(* Schneider Machine Expert - Basic project ControlPlantaCuchildeo, file version 2.6.0.0 *)
(* CompanyInformations: Name=DMA ENERGIA *)
(* ProjectInformations: Name=CONTROL POSICION SERVO, Description=Cuchildeo *)

HARDWARE
  Cpu 0: TM221CE40T
  ModuleExtensionObject 0: TM3AM6/G
  EthernetConfiguration: NetworkName=M221, IpAllocationMode=FixedAddress, IpAddress=192.168.10.132, SubnetMask=255.255.255.0
  SerialLineConfiguration: Baud=Baud19200, Parity=ParityEven, DataBits=DataBits8, StopBits=StopBits1, PhysicalMedium=PhysicalMediumRs485, SlaveId=1, Addressing=SlaveAddressing
  MastTask: UsePeriodScanMode=false, PeriodScan=100
  FastTask: Period=255
  CpuBehavior: StartingMode=StartAutoRunForced, AutoSaveRamOnEeprom=true, WatchdogPeriod=250

SYMBOLS  (address, symbol, comment, settings)
  %M0       CONTROL_MODE
  %M1       DIRECCION  "Direccion"
  %M2       SOBREVELOCIDAD1  "Limite velocidad 1"
  %M3       SOBREVELOCIDAD2  "Limite velocidad 2"
  %M4       OPERANDO_EN_VACIO
  %M5       OPEN_SETPOINT
  %M6       CONTROL_FREC
  %M7       CONTROL_POT
  %M8       SET_APERTURA
  %M9       GENERADOR
  %M10      MANUAL
  %M11      SET_CIERRE
  %M12      SOBREACELERACION
  %M13      TIMER
  %M14      BANDA_MUERTA
  %M15      CICLO_BOMBA1
  %M16      CICLO_BOMBA2
  %M17      C4_STOP
  %M18      AUX_ACELERACION
  %M19      ALM_SOBREACC
  %M20      C4_AL_GMOTOR
  %M21      DERECHA
  %M22      IZQUIERDA
  %M23      STOP
  %M24      TIMERON
  %M25      TIMEROFF
  %M26      C6_PUL_SUBIR
  %M27      C6_STOP
  %M28      ACELERACION
  %M29      AUX_ACC
  %M30      RESET_TIMER
  %M31      C5_PUL_POSICION
  %M32      C5_POSICIONANDO
  %M33      C5_ORDEN_SUBIR
  %M34      C5_ORDEN_BAJAR
  %M35      C2_PUL_POSICION
  %M36      C2_POSICIONANDO
  %M37      C2_ORDEN_SUBIR
  %M38      C2_ORDEN_BAJAR
  %M39      C1_INTERMEDIA
  %M40      C2_INTERMEDIA
  %M41      C3_INTERMEDIA
  %M42      C4_INTERMEDIA
  %M43      C5_INTERMEDIA
  %M44      C6_INTERMEDIA
  %M45      C5_PUL_STOP
  %M46      C2_PUL_STOP
  %M47      C1_TPO_ON_SUBIR
  %M48      C1_TPO_ON_BAJAR
  %M49      C2_TPO_ON_SUBIR
  %M50      C2_TPO_ON_BAJAR
  %M51      C3_TPO_ON_SUBIR
  %M52      C3_TPO_ON_BAJAR
  %M53      C4_TPO_ON_SUBIR
  %M54      C4_TPO_ON_BAJAR
  %M55      C5_TPO_ON_SUBIR
  %M56      C5_TPO_ON_BAJAR
  %M57      C6_TPO_ON_SUBIR
  %M58      C6_TPO_ON_BAJAR
  %M300     R_C1_PUL_SUBIR
  %M301     R_C1_STOP
  %M302     R_C1_PUL_BAJAR
  %M307     R_C2_STOP
  %M311     R_C3_PUL_SUBIR
  %M312     R_C3_STOP
  %M313     R_C3_PUL_BAJAR
  %M316     R_C4_PUL_SUBIR
  %M317     R_C4_STOP
  %M318     R_C4_PUL_BAJAR
  %M322     R_C5_STOP
  %M326     R_C6_PUL_SUBIR
  %M327     R_C6_STOP
  %M331     R_C5_PUL_POSICION
  %M335     R_C2_PUL_POSICION
  %S12      SB_RUNMODE  "El controlador se está ejecutando"
  %MW0      AUX_SET
  %MW1      SALIDA_CONTROL
  %MW2      MEDICION_APERTURA
  %MW3      PID0
  %MW4      SEÑAL_PV
  %MW5      ERROR_FREC
  %MW6      PV_SET
  %MW7      POT_SETEADA
  %MW8      PID1
  %MW9      POT_MEDIDA
  %MW10     GANANCIA_SETFREC
  %MW11     GANANCIA_SETPOT
  %MW12     KP
  %MW13     KI
  %MW14     KD
  %MW15     KPV
  %MW16     KIV
  %MW17     SALIDA_PI_VEL
  %MW18     RPM
  %MW19     SET_RPM
  %MW100    PEPE
  %MD0      SET
  %MD1      SET_FRECUENCIA
  %MD5      ERROR_FRECUENCIA
  %MD100    C2F_ALTURA
  %MD200    FREC_GEN
  %TM0      RETARDO  [Preset=2, Base=OneSecond]
  %TM1      RETARDO2  [Preset=1, Base=OneSecond]
  %TM2      RETARDO3  [Preset=10, Base=OneMilliSeconds]
  %TM3      TPO_CAMBIO_BOMBA2  [Preset=2880]
  %TM4      BANDAM  [Preset=100, Base=OneMilliSeconds, IsRetentive=true]
  %TM5      TPO_SOBRE_VEL1  [Preset=4, Base=OneSecond]
  %TM6      TPO_SOBRE_VEL2  [Preset=2, Base=OneSecond]
  %TM7      TPO_SOBRE_ACC  [Type=TOF, Preset=15, Base=OneSecond]
  %TM8      C5_TPO_MAX_SUBIR  [Preset=30, Base=OneSecond]
  %TM9      C5_TPO_MAX_BAJAR  [Preset=30, Base=OneSecond]
  %TM10     C6_TPO_MAX_SUBIR  [Preset=30, Base=OneSecond]
  %TM11     C6_TPO_MAX_BAJAR  [Preset=30, Base=OneSecond]
  %C0         [Preset=22]
  %SC0        "OPEN_VALUE"
  %I0.0     TURBINE_SPEED
  %I0.1     TURBINE_START_STOP
  %I0.2     AUTO_MANUAL
  %I0.3     OPEN_RISE
  %I0.4     OPEN_LOWER
  %I0.5     OPEN_
  %I0.6     GOV_RESET
  %I0.7     HIGH_PRESSURE
  %I0.8     LOW_PRESSURE
  %I0.9     RESET
  %I0.10    UNLOAD_VALVE_OPEN
  %I0.11    OIL_LEVEL_ALARM
  %I0.12    SPARE1
  %I0.13    SPARE2
  %Q0.0     PV_ON_OFF
  %Q0.1     VALVE_RP1_VENT_CONTROL
  %Q0.2     PUMP2_START_ORDER
  %Q0.3     VALVE_RP2_VENT_CONTROL
  %Q0.4     PUMP1_RUNNING
  %Q0.5     PUMP1_FAIL
  %Q0.6     PUMP2_RUNNING
  %Q0.7     PUMP2_FAIL
  %Q0.8     HPU_FAIL_OUTPUT
  %Q0.9     ARRANQUE
  %IW0.0    HPU_PRESSURE  [Type=Type_0_10V, Scope=Scope_Normal, Minimum=0, Maximum=1000]
  %IW0.1    HPU_OIL_TEMP  [Type=Type_0_10V, Scope=Scope_Normal, Minimum=0, Maximum=1000]
  %HSC0       [Type=FrequencyMeter, Preset=0, UseDoubleWord=true, DedicatedInputs(DedicatedInput(Activated=true)), ReflexOutputs(ReflexOutput(Activated=false, LessThanS0=false, GreaterOrEqualThanS0=true, GreaterOrEqualThanS1=false), ReflexOutput(Activated=false, LessThanS0=false, GreaterOrEqualThanS0=false, GreaterOrEqualThanS1=true)), Thresholds(Threshold(ThresholdType=NotUsed, Priority=7), Threshold(ThresholdT]
  %IW1.0      "Sensor"  [Type=Type_4_20mA, Scope=Scope_Customized, Minimum=4, Maximum=20]
  %IW1.1    REALIMENTACION  "Potenciometro"  [Type=Type_4_20mA, Scope=Scope_Customized, Minimum=4000, Maximum=20000]
  %QW1.0    PV  [Type=Type_0_10V, Scope=Scope_Customized, Minimum=0, Maximum=10000]
  %QW1.1    VAR_VEL  [Type=Type_4_20mA, Scope=Scope_Customized, Minimum=400, Maximum=2000]

POU Nuevo POU
  (* SectionNumber=1 *)

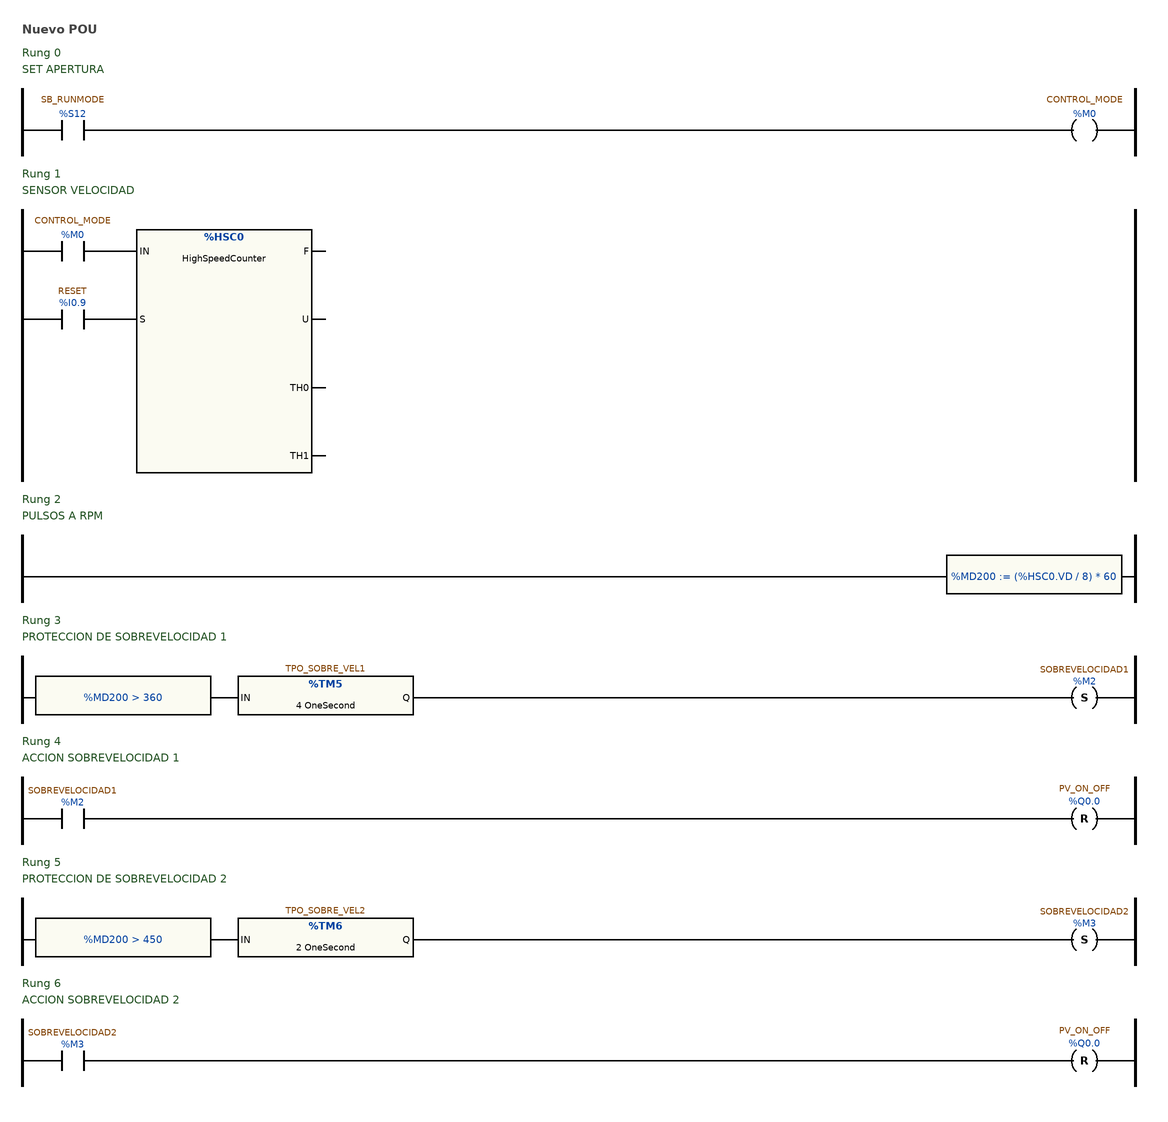

// Rung 0
// SET APERTURA
  LD %S12                 (* SB_RUNMODE *)
  ST %M0                  (* CONTROL_MODE *)
  // as ST:
  //   CONTROL_MODE := SB_RUNMODE;

// Rung 1
// SENSOR VELOCIDAD
  BLK %HSC0
  LD %M0                  (* CONTROL_MODE *)
  IN
  LD %I0.9                (* RESET *)
  S
  END_BLK
  // as ST:
  //   %HSC0(IN := CONTROL_MODE, S := RESET);

// Rung 2
// PULSOS A RPM
  LD 1
  [ %MD200 := ( %HSC0.VD / 8 ) * 60 ](* FREC_GEN *)
  // as ST:
  //   FREC_GEN := ( %HSC0.VD / 8 ) * 60;

// Rung 3
// PROTECCION DE SOBREVELOCIDAD 1
  BLK %TM5                (* TPO_SOBRE_VEL1 *)
  LD [ %MD200 > 360 ]     (* FREC_GEN *)
  IN
  OUT_BLK
  LD Q
  S %M2                   (* SOBREVELOCIDAD1 *)
  END_BLK
  // as ST:
  //   TPO_SOBRE_VEL1(IN := FREC_GEN > 360);
  //   IF TPO_SOBRE_VEL1.Q THEN SOBREVELOCIDAD1 := TRUE; END_IF;

// Rung 4
// ACCION SOBREVELOCIDAD 1
  LD %M2                  (* SOBREVELOCIDAD1 *)
  R %Q0.0                 (* PV_ON_OFF *)
  // as ST:
  //   IF SOBREVELOCIDAD1 THEN PV_ON_OFF := FALSE; END_IF;

// Rung 5
// PROTECCION DE SOBREVELOCIDAD 2
  BLK %TM6                (* TPO_SOBRE_VEL2 *)
  LD [ %MD200 > 450 ]     (* FREC_GEN *)
  IN
  OUT_BLK
  LD Q
  S %M3                   (* SOBREVELOCIDAD2 *)
  END_BLK
  // as ST:
  //   TPO_SOBRE_VEL2(IN := FREC_GEN > 450);
  //   IF TPO_SOBRE_VEL2.Q THEN SOBREVELOCIDAD2 := TRUE; END_IF;

// Rung 6
// ACCION SOBREVELOCIDAD 2
  LD %M3                  (* SOBREVELOCIDAD2 *)
  R %Q0.0                 (* PV_ON_OFF *)
  // as ST:
  //   IF SOBREVELOCIDAD2 THEN PV_ON_OFF := FALSE; END_IF;

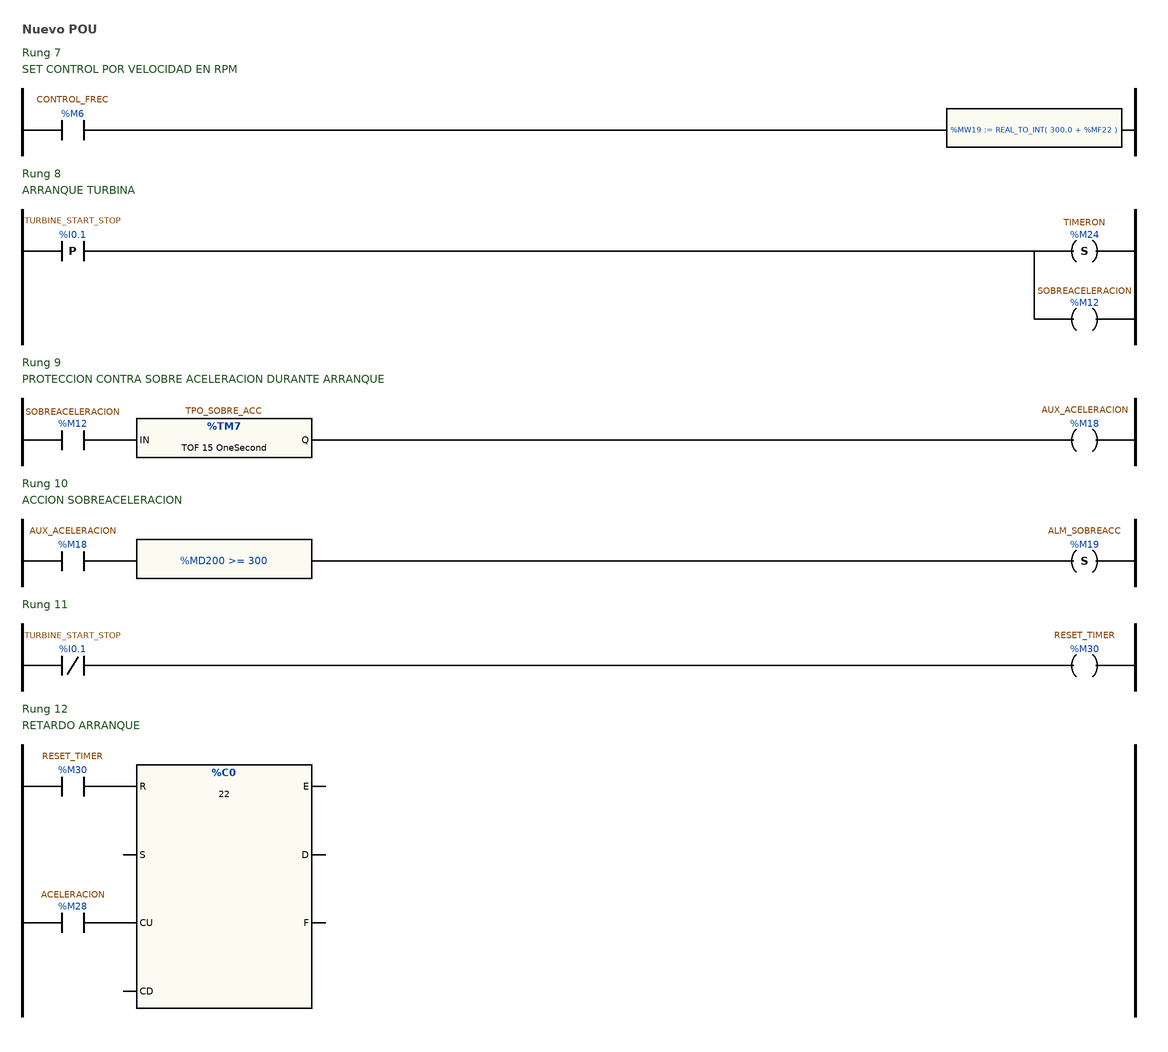

// Rung 7
// SET CONTROL POR VELOCIDAD EN RPM
  LD %M6                  (* CONTROL_FREC *)
  [ %MW19 := REAL_TO_INT ( 300.0 + %MF22 ) ](* SET_RPM *)
  // as ST:
  //   IF CONTROL_FREC THEN SET_RPM := REAL_TO_INT ( 300.0 + %MF22 ); END_IF;

// Rung 8
// ARRANQUE TURBINA
  LDR %I0.1               (* TURBINE_START_STOP *)
  S %M24                  (* TIMERON *)
  ST %M12                 (* SOBREACELERACION *)
  // as ST:
  //   IF RISING(TURBINE_START_STOP) THEN TIMERON := TRUE; END_IF;
  //   SOBREACELERACION := RISING(TURBINE_START_STOP);

// Rung 9
// PROTECCION CONTRA SOBRE ACELERACION DURANTE ARRANQUE
  BLK %TM7                (* TPO_SOBRE_ACC *)
  LD %M12                 (* SOBREACELERACION *)
  IN
  OUT_BLK
  LD Q
  ST %M18                 (* AUX_ACELERACION *)
  END_BLK
  // as ST:
  //   TPO_SOBRE_ACC(IN := SOBREACELERACION);
  //   AUX_ACELERACION := TPO_SOBRE_ACC.Q;

// Rung 10
// ACCION SOBREACELERACION
  LD %M18                 (* AUX_ACELERACION *)
  AND [ %MD200 >= 300 ]   (* FREC_GEN *)
  S %M19                  (* ALM_SOBREACC *)
  // as ST:
  //   IF AUX_ACELERACION AND FREC_GEN >= 300 THEN ALM_SOBREACC := TRUE; END_IF;

// Rung 11
  LDN %I0.1               (* TURBINE_START_STOP *)
  ST %M30                 (* RESET_TIMER *)
  // as ST:
  //   RESET_TIMER := NOT TURBINE_START_STOP;

// Rung 12
// RETARDO ARRANQUE
  BLK %C0
  LD %M30                 (* RESET_TIMER *)
  R
  LD %M28                 (* ACELERACION *)
  CU
  END_BLK
  // as ST:
  //   %C0(R := RESET_TIMER, CU := ACELERACION);

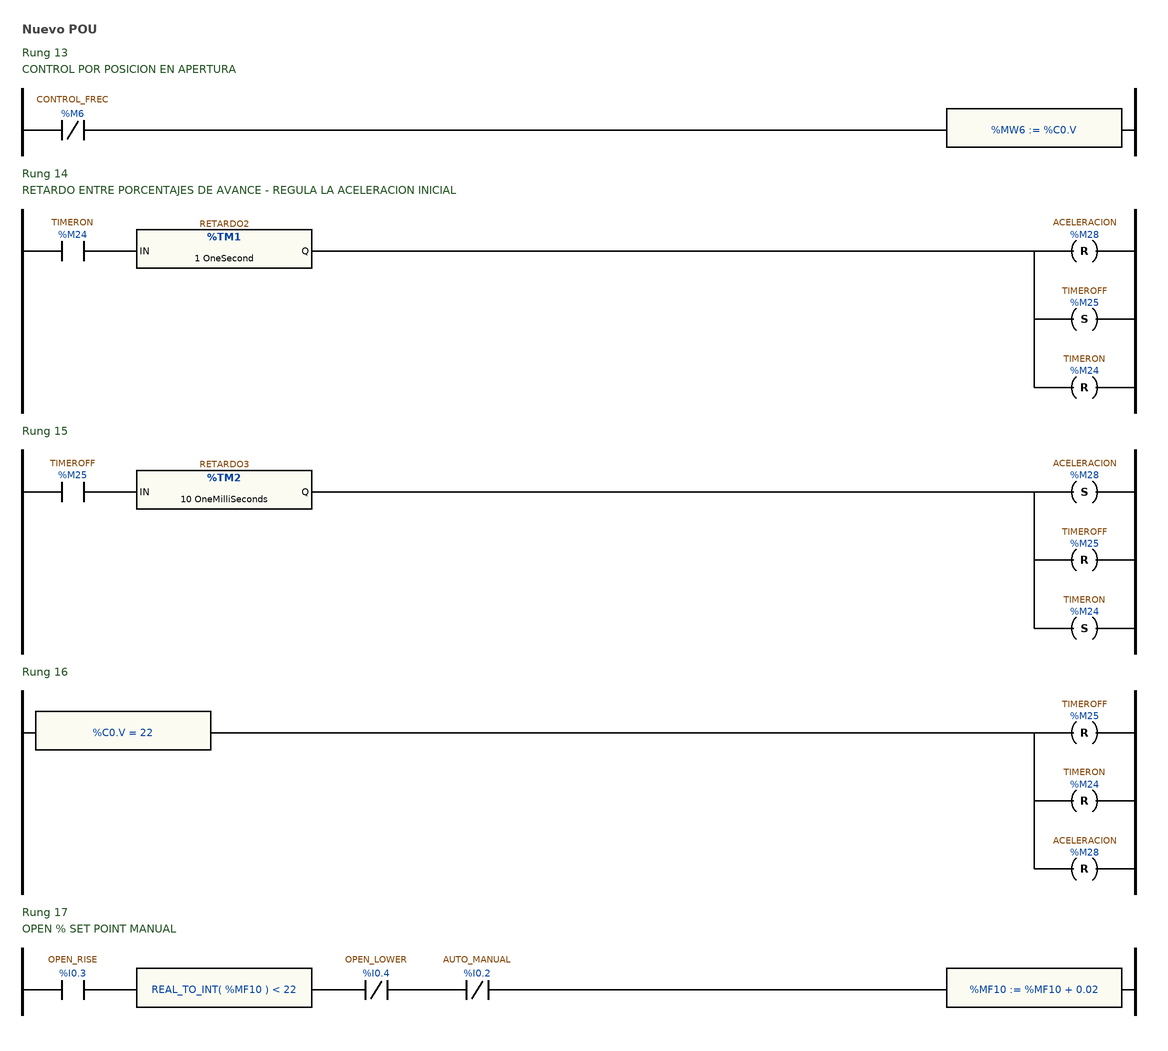

// Rung 13
// CONTROL POR POSICION EN APERTURA
  LDN %M6                 (* CONTROL_FREC *)
  [ %MW6 := %C0.V ]       (* PV_SET *)
  // as ST:
  //   IF NOT CONTROL_FREC THEN PV_SET := %C0.V; END_IF;

// Rung 14
// RETARDO ENTRE PORCENTAJES DE AVANCE - REGULA LA ACELERACION INICIAL
  BLK %TM1                (* RETARDO2 *)
  LD %M24                 (* TIMERON *)
  IN
  OUT_BLK
  LD Q
  R %M28                  (* ACELERACION *)
  S %M25                  (* TIMEROFF *)
  R %M24                  (* TIMERON *)
  END_BLK
  // as ST:
  //   RETARDO2(IN := TIMERON);
  //   IF RETARDO2.Q THEN ACELERACION := FALSE; END_IF;
  //   IF RETARDO2.Q THEN TIMEROFF := TRUE; END_IF;
  //   IF RETARDO2.Q THEN TIMERON := FALSE; END_IF;

// Rung 15
  BLK %TM2                (* RETARDO3 *)
  LD %M25                 (* TIMEROFF *)
  IN
  OUT_BLK
  LD Q
  S %M28                  (* ACELERACION *)
  R %M25                  (* TIMEROFF *)
  S %M24                  (* TIMERON *)
  END_BLK
  // as ST:
  //   RETARDO3(IN := TIMEROFF);
  //   IF RETARDO3.Q THEN ACELERACION := TRUE; END_IF;
  //   IF RETARDO3.Q THEN TIMEROFF := FALSE; END_IF;
  //   IF RETARDO3.Q THEN TIMERON := TRUE; END_IF;

// Rung 16
  LD [ %C0.V = 22 ]
  R %M25                  (* TIMEROFF *)
  R %M24                  (* TIMERON *)
  R %M28                  (* ACELERACION *)
  // as ST:
  //   IF %C0.V = 22 THEN TIMEROFF := FALSE; END_IF;
  //   IF %C0.V = 22 THEN TIMERON := FALSE; END_IF;
  //   IF %C0.V = 22 THEN ACELERACION := FALSE; END_IF;

// Rung 17
// OPEN % SET POINT MANUAL
  LD %I0.3                (* OPEN_RISE *)
  AND [ REAL_TO_INT ( %MF10 ) < 22 ]
  ANDN %I0.4              (* OPEN_LOWER *)
  ANDN %I0.2              (* AUTO_MANUAL *)
  [ %MF10 := %MF10 + 0.02 ]
  // as ST:
  //   IF OPEN_RISE AND REAL_TO_INT ( %MF10 ) < 22 AND NOT OPEN_LOWER AND NOT AUTO_MANUAL THEN %MF10 := %MF10 + 0.02; END_IF;

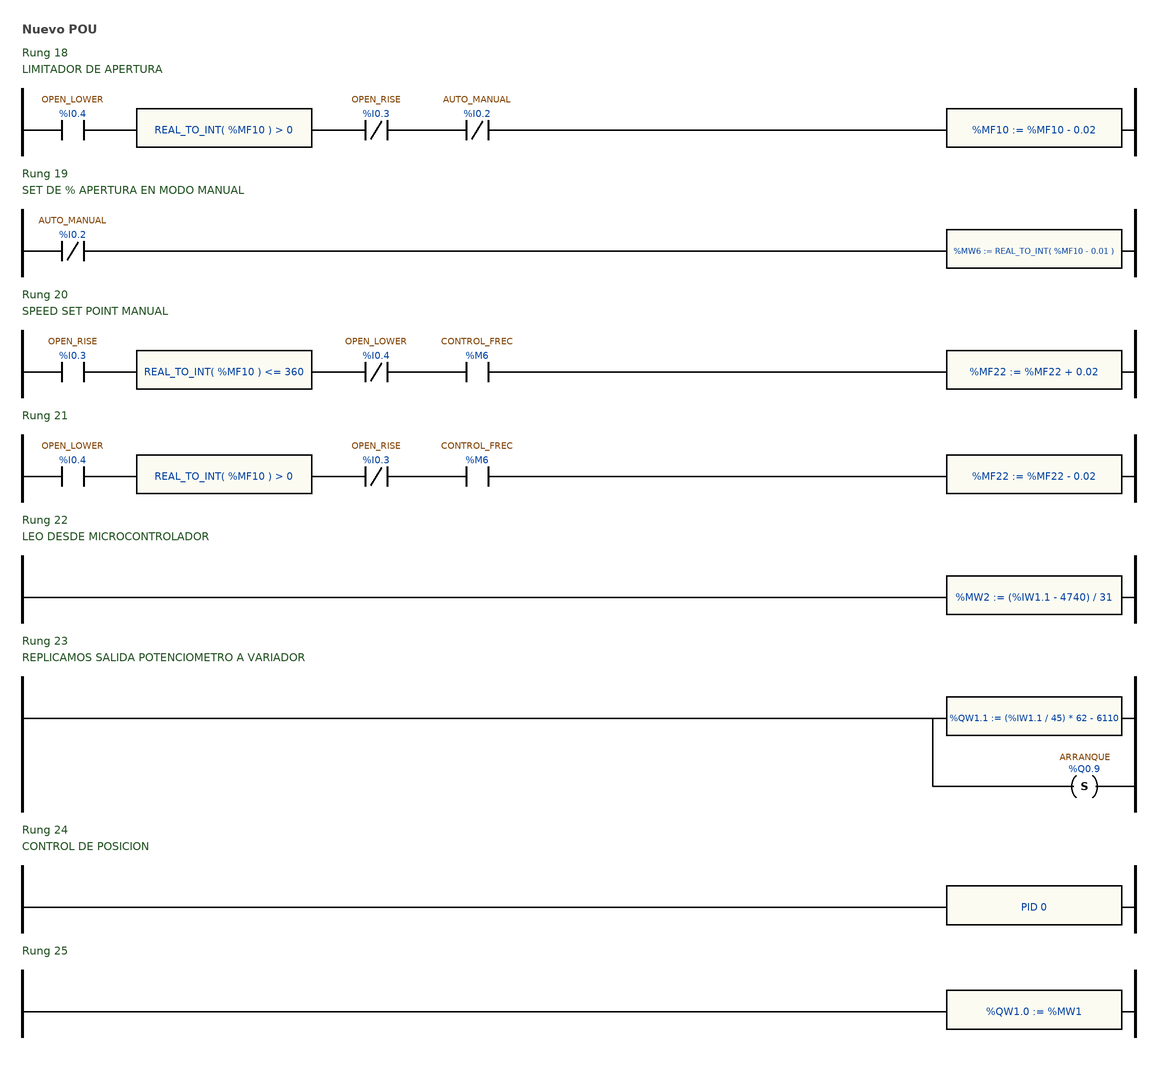

// Rung 18
// LIMITADOR DE APERTURA
  LD %I0.4                (* OPEN_LOWER *)
  AND [ REAL_TO_INT ( %MF10 ) > 0 ]
  ANDN %I0.3              (* OPEN_RISE *)
  ANDN %I0.2              (* AUTO_MANUAL *)
  [ %MF10 := %MF10 - 0.02 ]
  // as ST:
  //   IF OPEN_LOWER AND REAL_TO_INT ( %MF10 ) > 0 AND NOT OPEN_RISE AND NOT AUTO_MANUAL THEN %MF10 := %MF10 - 0.02; END_IF;

// Rung 19
// SET DE % APERTURA EN MODO MANUAL
  LDN %I0.2               (* AUTO_MANUAL *)
  [ %MW6 := REAL_TO_INT ( %MF10 - 0.01 ) ](* PV_SET *)
  // as ST:
  //   IF NOT AUTO_MANUAL THEN PV_SET := REAL_TO_INT ( %MF10 - 0.01 ); END_IF;

// Rung 20
// SPEED SET POINT MANUAL
  LD %I0.3                (* OPEN_RISE *)
  AND [ REAL_TO_INT ( %MF10 ) <= 360 ]
  ANDN %I0.4              (* OPEN_LOWER *)
  AND %M6                 (* CONTROL_FREC *)
  [ %MF22 := %MF22 + 0.02 ]
  // as ST:
  //   IF OPEN_RISE AND REAL_TO_INT ( %MF10 ) <= 360 AND NOT OPEN_LOWER AND CONTROL_FREC THEN %MF22 := %MF22 + 0.02; END_IF;

// Rung 21
  LD %I0.4                (* OPEN_LOWER *)
  AND [ REAL_TO_INT ( %MF10 ) > 0 ]
  ANDN %I0.3              (* OPEN_RISE *)
  AND %M6                 (* CONTROL_FREC *)
  [ %MF22 := %MF22 - 0.02 ]
  // as ST:
  //   IF OPEN_LOWER AND REAL_TO_INT ( %MF10 ) > 0 AND NOT OPEN_RISE AND CONTROL_FREC THEN %MF22 := %MF22 - 0.02; END_IF;

// Rung 22
// LEO DESDE MICROCONTROLADOR
  LD 1
  [ %MW2 := ( %IW1.1 - 4740 ) / 31 ](* MEDICION_APERTURA, REALIMENTACION *)
  // as ST:
  //   MEDICION_APERTURA := ( REALIMENTACION - 4740 ) / 31;

// Rung 23
// REPLICAMOS SALIDA POTENCIOMETRO A VARIADOR
  LD 1
  [ %QW1.1 := ( %IW1.1 / 45 ) * 62 - 6110 ](* VAR_VEL, REALIMENTACION *)
  S %Q0.9                 (* ARRANQUE *)
  // as ST:
  //   VAR_VEL := ( REALIMENTACION / 45 ) * 62 - 6110;
  //   ARRANQUE := TRUE;

// Rung 24
// CONTROL DE POSICION
  LD 1
  [ PID 0 ]
  // as ST:
  //   PID 0;

// Rung 25
  LD 1
  [ %QW1.0 := %MW1 ]      (* PV, SALIDA_CONTROL *)
  // as ST:
  //   PV := SALIDA_CONTROL;

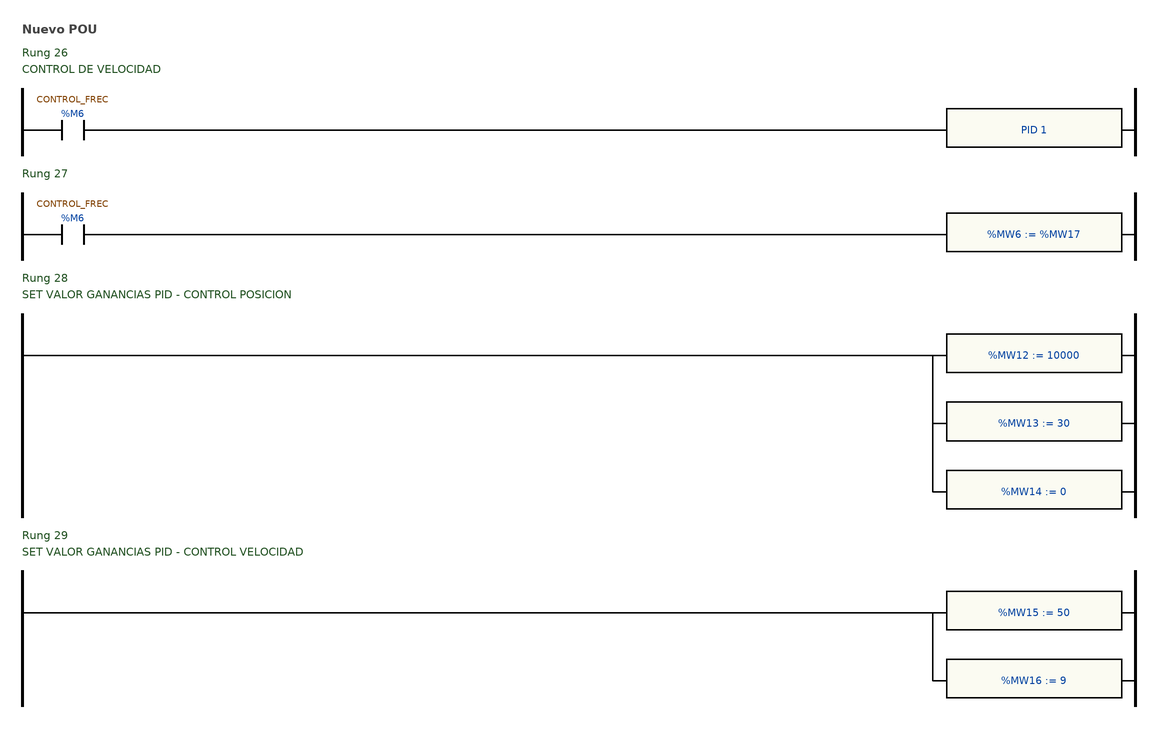

// Rung 26
// CONTROL DE VELOCIDAD
  LD %M6                  (* CONTROL_FREC *)
  [ PID 1 ]
  // as ST:
  //   IF CONTROL_FREC THEN PID 1; END_IF;

// Rung 27
  LD %M6                  (* CONTROL_FREC *)
  [ %MW6 := %MW17 ]       (* PV_SET, SALIDA_PI_VEL *)
  // as ST:
  //   IF CONTROL_FREC THEN PV_SET := SALIDA_PI_VEL; END_IF;

// Rung 28
// SET VALOR GANANCIAS PID - CONTROL POSICION
  LD 1
  [ %MW12 := 10000 ]      (* KP *)
  [ %MW13 := 30 ]         (* KI *)
  [ %MW14 := 0 ]          (* KD *)
  // as ST:
  //   KP := 10000;
  //   KI := 30;
  //   KD := 0;

// Rung 29
// SET VALOR GANANCIAS PID - CONTROL VELOCIDAD
  LD 1
  [ %MW15 := 50 ]         (* KPV *)
  [ %MW16 := 9 ]          (* KIV *)
  // as ST:
  //   KPV := 50;
  //   KIV := 9;
